VAR_GLOBAL CONSTANT
	cOversamples	: UINT := 1;					// number of oversamples
	cSamplingRate	: UINT := 100 * cOversamples;	// samplerate
END_VAR

(* stored: Version 1.1.0.1, ProductVersion 3.1.4026.17
   GVL Global_Constants: Id {9757b3a2-696e-42e1-9d86-e6fac84a7d73} *)
